# B&R Automation Studio project CaseWeek_user
Automation Studio 4.12.8.41 SP; technology packages: mapp 5.24.5, mappView 5.24.5

## Configuration X20CP1584

CPU X20CP1584, AutomationRuntime J4.93, Build 4.1.2, Safety 0.0, Vc V4.34.3

### Task classes (Cpu.sw)
```
Cyclic#1:
  ClockSigna <- Wizualizacja.ClockSignal.prg
Cyclic#4:
  Operation <- Sterowanie.Operation.prg
  Tanks <- Sterowanie.Tanks.prg
Binaries: mvLoader, TCLang, OpcUaSrv, udbdef, TCData, User, arconfig, sysconf, iomap, asfw, ashwac, ashwd, Role
Libraries: standard, astime, arssl, asieccon, fileio, runtime, AsBrStr
```

### Hardware
```
X20CP1584 : X20CP1584 v1.10.0.0
  Connector IF2:
    ActivateDevice = 1
  Connector IF3:
    DNAConfiguration = manual
  ConfigurationID = CaseWeek_user_X20CP1584
  UserPartitionSize = 0
  Simulation = 1
  TimerDeviceType = EPLX2X
  TimerDevice = X20CP1584.IF6
  TaskClassIdleTime = 2000
  FileDevice1
  FileDeviceName1 = Location
  FileDevicePath1 = C:\Temp\
  ActivateOpcUa = 1
  OpcUaInformationModels_PV_Version = 1
```

### Config.mpalarmxcore - X20CP1584/mappServices/Config.mpalarmxcore
```
Element gAlarmXCore (Type=mpalarmxcore)
  mapp.AlarmX.Core.Configuration:
    [0]:
      Name = LvLTank1IsTooHigh
      Message = Fluid level in tank 1 is above 80%!
      Behavior = PersistentAlarm
    [1]:
      Name = LvLTank2IsTooHigh
      Message = Fluid level in tank 2 is above 80%!
      Code = 1
      Behavior = PersistentAlarm
    [2]:
      Name = PressureTank1TooHigh
      Message = Pressure in tank 1 is too high!
      Code = 2
      Behavior = PersistentAlarm
    [3]:
      Name = PressureTank2TooHigh
      Message = Pressure in tank 2 is too high!
      Code = 3
      Behavior = PersistentAlarm
    [4]:
      Name = PressureTank1TooLow
      Message = Pressure in tank 1 is too low!
      Code = 4
      Behavior = PersistentAlarm
    [5]:
      Name = PressureTank2TooLow
      Message = Pressure in tank 2 is too low!
      Code = 5
      Behavior = PersistentAlarm
    [6]:
      Name = LvLTank3IsTooHigh
      Message = Fluid level in tank 3 is above 80%!
      Code = 6
      Behavior = PersistentAlarm
```

## Logical view

Binary libraries used (declarations not repeated): operator, runtime, astime, AsIecCon, standard, AsBrStr

### Global.var - Global variables
```iecst
VAR
	StartButton : BOOL;
	MixButton : BOOL;
	StopButton : BOOL;
END_VAR
```

### Package Logical/Libraries - Global libraries

- Visualisation Logical/mappView (not shown)

### Program Logical/Sterowanie/Operation (IEC)

#### Types.typ
```iecst
TYPE
	StepEnum :
		(
		STEP_START,
		STEP_FILL12,
		STEP_EMPTY12,
		STEP_FILL3,
		STEP_EMPTY3,
		STEP_MIX
		);
	ControlType : 	STRUCT
		Step : StepEnum;
	END_STRUCT;
	TankLvl : 	STRUCT
		zb1 : USINT;
		zb2 : USINT;
		zb3 : USINT;
	END_STRUCT;
	AnalogValue : 	STRUCT
		ValveRight : USINT;
		ValveLeft : USINT;
	END_STRUCT;
	CurrentTask : 	STRUCT
		Start : USINT;
		Stop : USINT;
		Nalewanie : USINT;
		Mieszanie : USINT;
	END_STRUCT;
END_TYPE
```

#### Variables.var
```iecst
VAR
	Control : ControlType;
	Tank : TankLvl;
	TimerMix : TON;
END_VAR
VAR CONSTANT
	Full : UINT := 10000;
END_VAR
VAR
	AnalogValve : AnalogValue;
END_VAR
```

#### Main.st
```iecst
PROGRAM _INIT
	gZb1_poziom;
	gZb1_zawor;
	gZb2_poziom;
	gZb2_zawor;

	gZb3_poziom;
	gZb3_zawor_glowny;
	gZb3_zawor_lewy;
	gZb3_zawor_prawy;

	gMieszadlo;
	StartButton := FALSE;
	MixButton := FALSE;

	AnalogValve.ValveRight := 50;
	AnalogValve.ValveLeft := 50;
END_PROGRAM

PROGRAM _CYCLIC
	IF StopButton THEN
		StartButton := FALSE;
		Control.Step := STEP_START;
	END_IF;
	CASE Control.Step OF
		STEP_START:
			gZb1_zawor := FALSE;
			gZb2_zawor := FALSE;
			gZb3_zawor_prawy := FALSE;
			gZb3_zawor_lewy := FALSE;
			gZb3_zawor_glowny := FALSE;
			IF StartButton THEN
				Control.Step := STEP_FILL12;
			END_IF;

		STEP_FILL12:
			StartButton := FALSE;
			gZb1_zawor := TRUE;
			gZb2_zawor := TRUE;
			IF gZb1_poziom >=8000 AND gZb2_poziom >= 8000 THEN
				Control.Step := STEP_EMPTY12;
			END_IF;

		STEP_EMPTY12:
			gZb1_zawor := FALSE;
			gZb2_zawor := FALSE;
			Control.Step := STEP_FILL3;

		STEP_FILL3:
			gZb3_zawor_prawy := AnalogValve.ValveRight;
			gZb3_zawor_lewy := AnalogValve.ValveLeft;
			IF gZb3_poziom >=8000 AND gMieszadlo = FALSE THEN
				gZb3_zawor_prawy := FALSE;
				gZb3_zawor_lewy := FALSE;
				Control.Step := STEP_EMPTY3;
			END_IF;
			IF gZb3_poziom = 10000 AND gMieszadlo = TRUE THEN
				gZb3_zawor_prawy := FALSE;
				gZb3_zawor_lewy := FALSE;
				Control.Step := STEP_MIX;
			END_IF;

		STEP_MIX:
			TimerMix.PT := T#5s;
			TimerMix.IN := TRUE;
			gMieszadlo := TRUE;
			IF TimerMix.Q = TRUE THEN
				TimerMix.IN := FALSE;
				gMieszadlo := FALSE;
				Control.Step := STEP_EMPTY3;
			END_IF;

		STEP_EMPTY3:
			gZb3_zawor_glowny := TRUE;
			IF gZb3_poziom = 0 THEN
				Control.Step := STEP_START;
			END_IF;
	END_CASE;

	Tank.zb1 := INT_TO_USINT((gZb1_poziom * 100) / Full);
	Tank.zb2 := INT_TO_USINT((gZb2_poziom * 100) / Full);
	Tank.zb3 := INT_TO_USINT((gZb3_poziom * 100) / Full);

	TimerMix();

END_PROGRAM

PROGRAM _EXIT
	(* Insert code here *)

END_PROGRAM
```

### Program Logical/Sterowanie/Alarm (IEC)

#### Variables.var
```iecst
VAR
	MpAlarmXCore_0 : MpAlarmXCore;
	PressureTank1 : REAL;
	PressureTank2 : REAL;
END_VAR
```

#### Main.st
```iecst
PROGRAM _INIT
	(* MpLink przekazujemy przez referencję ADR *)
	MpAlarmXCore_0(MpLink := ADR(gAlarmXCore), Enable := TRUE);
END_PROGRAM

PROGRAM _CYCLIC
	(* Można wywołać funkcję bez parametrów *)
	IF gZb1_poziom > 8000.0 THEN
		MpAlarmXSet(gAlarmXCore, 'LvLTank1IsTooHigh');
	END_IF;
	(* Nie podajemy MpLink do Set przez referencję *)

	IF gZb1_poziom < 8000.0 THEN
		MpAlarmXReset(gAlarmXCore, 'LvLTank1IsTooHigh');
	END_IF;

	IF gZb2_poziom > 8000.0 THEN
		MpAlarmXSet(gAlarmXCore, 'LvLTank2IsTooHigh');
	END_IF;

	IF gZb2_poziom < 8000.0 THEN
		MpAlarmXReset(gAlarmXCore, 'LvLTank2IsTooHigh');
	END_IF;

	IF gZb3_poziom > 8000.0 THEN
		MpAlarmXSet(gAlarmXCore, 'LvLTank3IsTooHigh');
	END_IF;

	IF gZb3_poziom < 8000.0 THEN
		MpAlarmXReset(gAlarmXCore, 'LvLTank3IsTooHigh');
	END_IF;
	//Pressure 1
	IF PressureTank1 > 4.0 THEN
		MpAlarmXSet(gAlarmXCore, 'PressureTank1TooHigh');
	END_IF;

	IF PressureTank1 < 4.0 THEN
		MpAlarmXReset(gAlarmXCore, 'PressureTank1TooHigh');
	END_IF;

	IF PressureTank1 > 2.0 THEN
		MpAlarmXReset(gAlarmXCore, 'PressureTank1TooLow');
	END_IF;

	IF PressureTank1 < 2.0 THEN
		MpAlarmXSet(gAlarmXCore, 'PressureTank1TooLow');
	END_IF;

	//Pressure 2
	IF PressureTank2 > 4.0 THEN
		MpAlarmXSet(gAlarmXCore, 'PressureTank2TooHigh');
	END_IF;

	IF PressureTank2 < 4.0 THEN
		MpAlarmXReset(gAlarmXCore, 'PressureTank2TooHigh');
	END_IF;

	IF PressureTank2 > 2.0 THEN
		MpAlarmXReset(gAlarmXCore, 'PressureTank2TooLow');
	END_IF;

	IF PressureTank2 < 2.0 THEN
		MpAlarmXSet(gAlarmXCore, 'PressureTank2TooLow');
	END_IF;

	MpAlarmXCore_0(MpLink := ADR(gAlarmXCore), Enable := TRUE);
END_PROGRAM

PROGRAM _EXIT
	(* W sekcji exit trzeba wywołać/wyłaczyć blok funkcyjny (Enable := FALSE) *)
	MpAlarmXCore_0(MpLink := ADR(gAlarmXCore), Enable := FALSE);
END_PROGRAM
```

### Program Logical/Sterowanie/Recipe (IEC)

#### Types.typ
```iecst
TYPE
	Recipe_Type : 	STRUCT
		AnalogValveRight : INT := 75;
		AnalogValveLeft : INT := 45;
		TankLevel1 : INT := 5700;
		TankLevel2 : INT := 6500;
		TankLevel3 : INT := 7800;
		MixerOn : BOOL := TRUE;
	END_STRUCT;
END_TYPE
```

#### Variables.var
```iecst
VAR
	Recipe : Recipe_Type;
	MpRecipeXml_0 : MpRecipeXml;
	MpRecipeRegPar_0 : MpRecipeRegPar; (*UI-Connection*)
	MpRecipeUI_0 : MpRecipeUI; (*MpRecipeUI for UI Connection to the ice cream machine*)
	UIConnect : MpRecipeUIConnectType; (*UI Connection - contains the parameters needed for the connection*)
	Save : BOOL;
	Load : BOOL;
END_VAR
```

#### Main.st
```iecst
PROGRAM _INIT
	(* Zapis przepisu do C:\Temp\ *)
	MpRecipeXml_0.Enable := TRUE;
	MpRecipeXml_0.MpLink := ADR(gRecipeXml);
	MpRecipeXml_0.DeviceName := ADR('Location');
	MpRecipeXml_0.FileName := ADR('Recipe');

	MpRecipeRegPar_0.Enable := TRUE;
	MpRecipeRegPar_0.MpLink := ADR(gRecipeXml);
	MpRecipeRegPar_0.PVName := ADR('Recipe:Recipe');

	MpRecipeUI_0.Enable := TRUE;
	MpRecipeUI_0.MpLink := ADR(gRecipeXml);
	MpRecipeUI_0.UIConnect := ADR(UIConnect);
END_PROGRAM

PROGRAM _CYCLIC
	(* Wywołanie bloków funkcyjnych *)
	MpRecipeXml_0();
	MpRecipeRegPar_0();
	MpRecipeUI_0();

	IF Save THEN
		MpRecipeXml_0.Load := FALSE;
		MpRecipeXml_0.Save := TRUE;
		Save := FALSE;
	END_IF;

	IF Load THEN
		MpRecipeXml_0.Save := FALSE;
		MpRecipeXml_0.Load := TRUE;
		Load := FALSE;
	END_IF;
END_PROGRAM

PROGRAM _EXIT
	(* Wyłączenie bloków funkcyjnych *)
	MpRecipeXml_0.Enable := FALSE;
	MpRecipeXml_0();

	MpRecipeRegPar_0.Enable := FALSE;
	MpRecipeRegPar_0();

	MpRecipeUI_0.Enable := FALSE;
	MpRecipeUI_0();
END_PROGRAM
```

Listed in the project but not available here: Logical/Global.typ, Logical/Wizualizacja, Logical/Sterowanie/mappingVariables.var, Logical/Sterowanie/Tanks
